FUNCTION_BLOCK Kulbana2
  (* Version 1.0, 2007-08-20, Goran Cengic, Chalmers *)
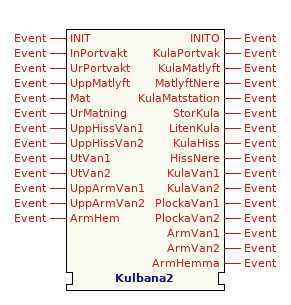
  EVENT_INPUT
    INIT;
    InPortvakt;
    UrPortvakt;
    UppMatlyft;
    Mat;
    UrMatning;
    UppHissVan1;
    UppHissVan2;
    UtVan1;
    UtVan2;
    UppArmVan1;
    UppArmVan2;
    ArmHem;
  END_EVENT
  EVENT_OUTPUT
    INITO;
    KulaPortvak;
    KulaMatlyft;
    MatlyftNere;
    KulaMatstation;
    StorKula;
    LitenKula;
    KulaHiss;
    HissNere;
    KulaVan1;
    KulaVan2;
    PlockaVan1;
    PlockaVan2;
    ArmVan1;
    ArmVan2;
    ArmHemma;
  END_EVENT
  VAR
    liten_kula : INT := 0;
  END_VAR
  EC_STATES
    START;
    INIT : -> INITO;
    STATE1 : -> KulaPortvakt;
    STATE2 : -> KulaMatlyft;
    STATE3 : -> KulaMatstation;
    STATE4 : StorKula -> StorKula;
    STATE5 : LitenKula -> LitenKula;
    STATE6 : -> KulaHiss, -> MatlyftNere;
    STATE7 : -> KulaVan1;
    STATE8 : -> KulaVan2;
    STATE9 : -> PlockaVan1, -> HissNere;
    STATE10 : -> PlockaVan2, -> HissNere;
    STATE11 : -> ArmVan1;
    STATE12 : -> ArmVan2;
    STATE13 : -> ArmHemma;
  END_STATES
  EC_TRANSITIONS
    START TO INIT := INIT;
    INIT TO START := 1;
    START TO STATE1 := InPortvakt;
    STATE1 TO START := 1;
    START TO STATE2 := UrPortvakt;
    STATE2 TO START := 1;
    START TO STATE3 := UppMatlyft;
    STATE3 TO START := 1;
    START TO STATE4 := Mat AND liten_kula = 0;
    STATE4 TO START := 1;
    START TO STATE5 := Mat AND liten_kula > 0;
    STATE5 TO START := 1;
    START TO STATE6 := UrMatning;
    STATE6 TO START := 1;
    START TO STATE7 := UppHissVan1;
    STATE7 TO START := 1;
    START TO STATE8 := UppHissVan2;
    STATE8 TO START := 1;
    START TO STATE9 := UtVan1;
    STATE9 TO START := 1;
    START TO STATE10 := UtVan2;
    STATE10 TO START := 1;
    START TO STATE11 := UppArmVan1;
    STATE11 TO START := 1;
    START TO STATE12 := UppArmVan2;
    STATE12 TO START := 1;
    START TO STATE13 := ArmHem;
    STATE13 TO START := 1;
  END_TRANSITIONS
  ALGORITHM StorKula IN Java:
liten_kula = (liten_kula + 1) % 3;
  END_ALGORITHM
  ALGORITHM LitenKula IN Java:
liten_kula = (liten_kula + 1) % 3;
  END_ALGORITHM
END_FUNCTION_BLOCK
